ABB RobotStudio station: IRB1600_20220607-170026.rsstn

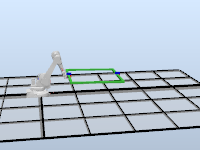
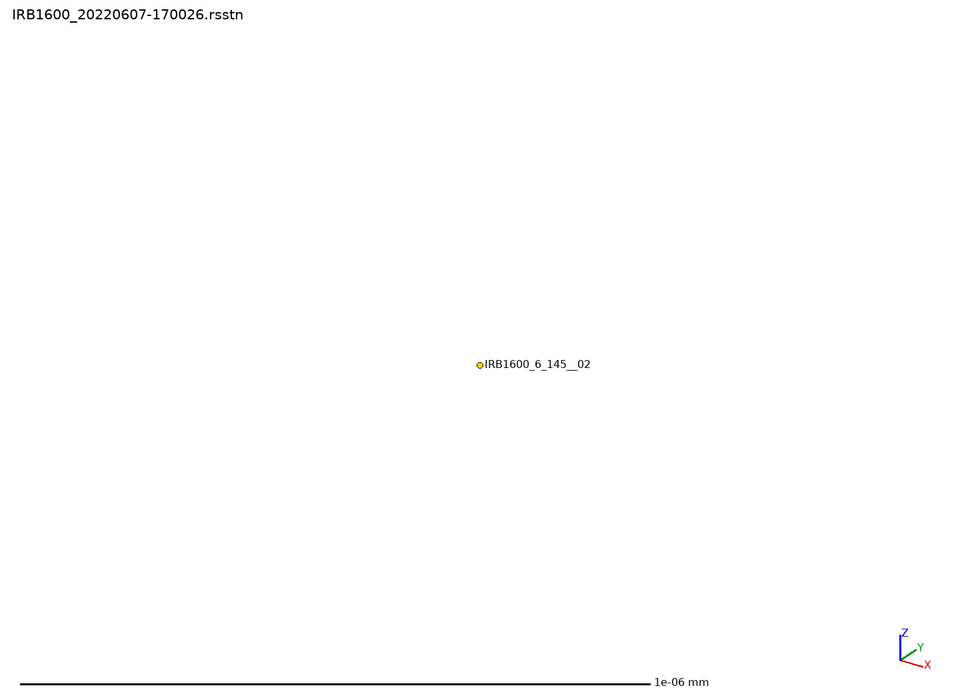
[picture v1: parts stored in the station drawn from their meshes, with robot base, taught points and paths (robot models come from the ABB library and are not in the file)]
Station Solution1 (saved by RobotStudio 21.2.9526.0)
Controller IRB1600_6_145
  mechanical unit ROB_1: IRB1600_6_145__02, 6 joints, base frame (0, 0, 0) mm
Layout (positions relative to the parent item):
  - IRB1600_6_145__02 [mechanism, from Robots\IRB1600_6_145_G_02.rslib] at (0, 0, 0) mm; joint values [0, 0.5566, 0.651, 0, -1.2175, 0] (rad or m)
  - surface [part] at (1555.48, 0, 522.35) mm, rotated rx 180 ry -1.79 rz 180 deg, size 1500 x 1500 x 50 mm
  - flange_connector [part, from Tools\IsoPlate_small_Binzel.rslib] at (797.97, 0, 520.65) mm, rotated rx 0 ry 89.43 rz 0 deg
  - Frame_3 [frame] at (844.92, 11.12, 1166.59) mm
  - Frame_4 [frame] at (2269.62, 18.76, 1121.91) mm
Attachment: flange_connector is attached to IRB1600_6_145__02 / Link6
Attachment: surface is attached to flange_connector
Targets, tools, work objects and paths stored in the station, written as RAPID:
! task T_ROB1
MODULE Module1
  LOCAL PERS wobjdata egm_wobj:=[FALSE,TRUE,"",[[0,0,0],[1,0,0,0]],[[0,0,0],[1,0,0,0]]];
  PROC main()
    EGM_CARTESIAN_MOVE;
  ENDPROC
  PROC EGM_CARTESIAN_MOVE()
    WaitTime 2;
  ENDPROC
ENDMODULE

! task T_ROB1
MODULE CalibData
  TASK PERS tooldata Tooldata_4:=[TRUE,[[0,0,0],[1,0,0,0]],[1,[0,0,1],[1,0,0,0],0,0,0]];
  TASK PERS tooldata Tooldata_5:=[TRUE,[[0,0,0],[1,0,0,0]],[1,[0,0,1],[1,0,0,0],0,0,0]];
  TASK PERS tooldata Tooldata_6:=[TRUE,[[0,0,0],[1,0,0,0]],[1,[0,0,1],[1,0,0,0],0,0,0]];
  TASK PERS tooldata Tooldata_7:=[TRUE,[[-23.772999999,2.161,40.120999999],[0.707106781,0,-0.707106781,0]],[1,[0,0,1],[1,0,0,0],0,0,0]];
  TASK PERS tooldata Tooldata_8:=[TRUE,[[35.292999999,18.761,1471.373000001],[0.707106781,0,-0.707106781,0]],[1,[0,0,1],[1,0,0,0],0,0,0]];
ENDMODULE

